FUNCTION_BLOCK FB_TankTest  EXTENDS FB_TestSuite
VAR_INPUT
END_VAR
VAR_OUTPUT
END_VAR
VAR
END_VAR

END_FUNCTION_BLOCK

(* stored: Version 1.1.0.1, ProductVersion 3.1.4024.16
   POU FB_TankTest: Id {2fba3182-35e4-45a1-b90b-c376c1549b6d}, SpecialFunc None *)
